Fanuc KAREL source: ko00150.KL

-- PROVISIONAL review KL for V940-1; original PC SHA256 d0c5de21ccd488a87f6b80332e29fe7ce07a5c46c8cd7665936d4c25e7a3505a
-- Incomplete behavior may be omitted. Consult companion uncertainty JSON. Do not deploy.
PROGRAM KO00150
%NOLOCKGROUP
VAR
  R : REAL
  N : REAL
-- UNRESOLVED_DECL CFG type=00001c
-- UNRESOLVED_DECL OUT type=000102
BEGIN
  -- V9_ZERO_TABLE_METADATA_HINT layout=0001; no indexed target words; source/name/runtime held
  -- UNRESOLVED_PC offsets 5-13; opcodes 9D,64,23
  -- UNRESOLVED_PC offsets 18-29; opcodes 2E,23
  -- UNRESOLVED_PC offsets 34-44; opcodes 9D,22,A5
  -- UNRESOLVED_PC offsets 49-106; opcodes 27,22,22,22,22,22,22,22,76,7E,4A
  -- UNRESOLVED_PC offsets 111-115; opcodes 7F
END KO00150
